TYPE T_CodeCRYPTO : STRING[20];
END_TYPE

(* stored: Version 1.1.0.1
   DUT T_CodeCRYPTO: Id {e60027c5-37c7-40a3-b130-a4c12797c47b} *)
